{attribute addProperty BoxType "EK1122-0000-0018"}
{attribute addProperty Id "Beckhoff_ER8xxxsub_EK1100EK1100_179A0949162A_0001_ER8309_1022_0018ER8309_7EF99CA440851"}
{attribute addProperty CRC "3328782902"}
{attribute addProperty SizeInBites "424"}
{attribute addProperty SizeInBytes "53"}
TYPE Beckhoff_ER8xxxEK1122_C6693236 EXTENDS EK1122_179A0949 :
STRUCT
	{attribute addProperty Name "Beckhoff_ER8xxxsub_EK1100"}
	Beckhoff_ER8xxxsub_EK1100 : EK1100_179A0949;
	{attribute addProperty Name "A_0001_ER8309_1022_0018"}
	A_0001_ER8309_1022_0018 : ER8309_7EF99CA4;
END_STRUCT
END_TYPE

(* stored: Version 1.2.0.0, ProductVersion 3.1.4024.9
   DUT Beckhoff_ER8xxxEK1122_C6693236: Id {c09d24f8-5d29-4afd-abd5-840cd93bf0d3} *)
